PROGRAM ManualControl
VAR
	
	MotorControl: MotorControl;
	R_TRIG_0: R_TRIG;
	R_TRIG_1: R_TRIG;
	R_TRIG_2: R_TRIG;
	R_TRIG_3: R_TRIG;
	TON_0: TON;
	SR_0: SR;
	
	Compressor_0: Compressor;
END_VAR

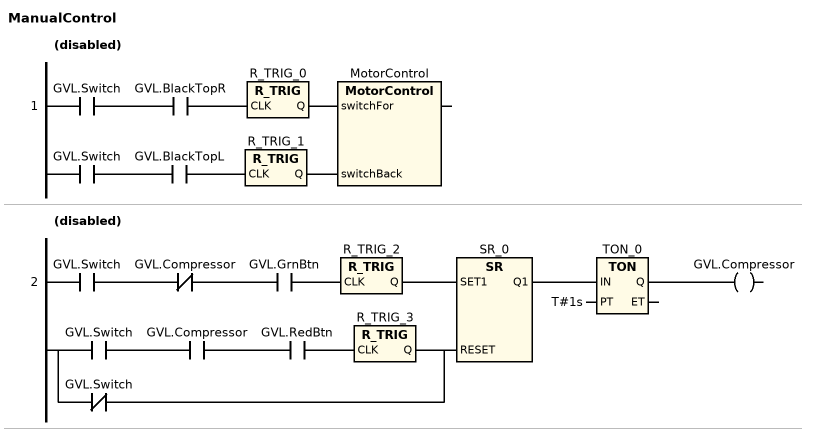
// NETWORK 1 (disabled)
// R_TRIG_0(CLK := GVL.Switch AND GVL.BlackTopR); // R_TRIG
// R_TRIG_1(CLK := GVL.Switch AND GVL.BlackTopL); // R_TRIG
// MotorControl(switchFor := R_TRIG_0.Q, switchBack := R_TRIG_1.Q);

// NETWORK 2 (disabled)
// R_TRIG_2(CLK := GVL.Switch AND NOT GVL.Compressor AND GVL.GrnBtn); // R_TRIG
// R_TRIG_3(CLK := GVL.Switch AND GVL.Compressor AND GVL.RedBtn); // R_TRIG
// SR_0(SET1 := R_TRIG_2.Q, RESET := R_TRIG_3.Q OR NOT GVL.Switch); // SR
// TON_0(IN := SR_0.Q1, PT := T#1s); // TON
// GVL.Compressor := TON_0.Q;

END_PROGRAM

(* stored: Version 1.1.0.1, ProductVersion 3.1.4024.12
   POU ManualControl: Id {5e8494a2-79e3-4126-acde-e6023512b35a}, SpecialFunc None *)
